// TIA Portal project "BOMBAS" (V15.1)

(* hardware
DEVICE "S7-1200 station_1"  S7-1200 Station
   slot 0: "Rack_0"  S7-1200 Rack  Rack  V1.0
   slot 1: "PLC_1"  CPU 1214C DC/DC/DC  6ES7 214-1AG40-0XB0  V4.2
DEVICE "HMI_1"  TP900 Comfort
   slot 0: "HMI_1"  TP900 Comfort  6AV2 124-0JC01-0AX0  15.1.0.0
   slot 1: "HMI_RT_1"  TP900 Comfort  6AV2 124-0JC01-0AX0  15.1.0.0
   slot 5: "HMI_1.IE_CP_1"  PROFINET Interface  15.0.1.0
      slot 1: "Interfaz PROFINET_1"  PROFINET Interface
         slot 1: "Port_1"  Port
         slot 2: "Port_2"  Port
   slot 7: "HMI_1.MPI/DP_CP_1"  MPI/DP Interface  15.0.1.0
*)

// ===== PLC "PLC_1"  CPU 1214C DC/DC/DC =====

VAR_GLOBAL   // PLC tag table "MODOS_ESTADOS"
   "HMI_PULSADOR_AUTOMATICO" AT %M2.1 : Bool;
   "HMI_PULSADOR_MANUAL" AT %M2.2 : Bool;
   "HMI_PULSADOR_STOP" AT %M2.3 : Bool;
   "ESTADO_MODO_MANUAL" AT %M2.4 : Bool;
   "ESTADO_MODO_AUTOMATICO" AT %M2.5 : Bool;
   "ESTADO_MODO_STOP" AT %M2.6 : Bool;
   "MODO_AUTOMATICO_START" AT %M2.7 : Bool;
   "HMI_PULSADOR_START" AT %M3.0 : Bool;
END_VAR

TYPE "BOMBA"
   STRUCT
      MOTOR : Bool;
      Tiempo_Total : UDInt;
      Tiempo_Acumulado : UDInt;
      Tiempo_Actual : UDInt;
      Tiempo_Trabajo : UDInt := 180;
   END_STRUCT;
END_TYPE

DATA_BLOCK "MAQUINA_ESTADO_BOMBAS_DB"   // DB1
{ S7_Optimized_Access := 'TRUE' }
VERSION : 0.1
// stored: InstanceOfName MAQUINA_ESTADO_BOMBAS
"MAQUINA_ESTADO_BOMBAS"
BEGIN
END_DATA_BLOCK

DATA_BLOCK "VARIABLES_GLOBALES"   // DB2
{ S7_Optimized_Access := 'TRUE' }
VERSION : 0.1
   VAR
      SALIDA_BOMBA_1 : "BOMBA";
      SALIDA_BOMBA_2 : "BOMBA";
      SALIDA_AUTOMATICO_BOMBA_1 : Bool;
      SALIDA_AUTOMATICO_BOMBA_2 : Bool;
      Tiempo_Cumplido_Bomba_1 : Bool;
      Tiempo_Cumplido_Bomba_2 : Bool;
      Tiempo_Formateado : Array[0..1] of Time_Of_Day;
      Numero_Str : String;
      HORA_STR : String;
      Tiempo_Bomba_1Str : String;
      Tiempo_Bomba_2Str : String;
      Variable_Ejemplo_VisualBasic : Int := 123;
      variable_string_visual : String := '123A';
      variable_string_visual2 : Array[0..2] of String;
      ejemplo_timeofdaytodint : DInt;
      tiempo : Time_Of_Day;
      Resultado_Conversion : Real;
   END_VAR
BEGIN
   SALIDA_BOMBA_1.Tiempo_Trabajo := 180;
   SALIDA_BOMBA_2.Tiempo_Trabajo := 180;
END_DATA_BLOCK

DATA_BLOCK "SALIDA_BOMBA_DB"   // DB3
{ S7_Optimized_Access := 'TRUE' }
VERSION : 0.1
// stored: InstanceOfName SALIDA_BOMBA
"SALIDA_BOMBA"
BEGIN
END_DATA_BLOCK

DATA_BLOCK "SALIDA_BOMBA_DB_1"   // DB5
{ S7_Optimized_Access := 'TRUE' }
VERSION : 0.1
// stored: InstanceOfName SALIDA_BOMBA
"SALIDA_BOMBA"
BEGIN
END_DATA_BLOCK

DATA_BLOCK "ALARMAS_DIAS"   // DB6
{ S7_Optimized_Access := 'TRUE' }
VERSION : 0.1
   VAR
      MOTORES : Array[1..3] of Struct
         DIA : Struct
            HORA_ACTIVACION : Array[1..7] of Time_Of_Day;
            HORA_DESACTIVACION : Array[1..7] of Time_Of_Day;
         END_STRUCT;
         ESTADO_MOTOR : Bool;
      END_STRUCT;
      HORA_ACTIVACION : Time_Of_Day;
      HORA_DESACTIVACION : Time_Of_Day;
   END_VAR
BEGIN
END_DATA_BLOCK

// folder: RELOJ

DATA_BLOCK "RELOJ_VARIABLES"   // DB4
{ S7_Optimized_Access := 'TRUE' }
VERSION : 0.1
   VAR
      HORA_ACTUAL : DTL;
      HORA_ANTERIOR : DTL;
      RET : Int;
      output_second : Bool;
   END_VAR
BEGIN
END_DATA_BLOCK

// folder: (top level)

FUNCTION_BLOCK "MAQUINA_ESTADO_BOMBAS"   // FB1, SCL
{ S7_Optimized_Access := 'TRUE' }
VERSION : 0.1
   VAR_INPUT
      ESTADO_AUTOMATICO : Bool;
      BOTON_START : Bool;
      BOTON_PARO_AUTOMATICO : Bool;
      Tiempo_Cumplido_Bomba_1 : Bool;
      Tiempo_Cumplido_Bomba_2 : Bool;
      BOTON_PARO_GENERAL : Bool;
      Tiempo_Bomba_1 : UDInt;
      Tiempo_Bomba_2 : UDInt;
   END_VAR
   VAR_OUTPUT
      MOTOR1 : Bool;
      MOTOR2 : Bool;
   END_VAR
   VAR
      ESTADO : USInt := 0;
   END_VAR
   VAR CONSTANT
      ESTADO_0 : USInt := 0;
      ESTADO_1 : USInt := 1;
      ESTADO_2 : USInt := 2;
      ESTADO_3 : USInt := 3;
      ESTADO_4 : USInt := 4;
      ESTADO_5 : USInt := 5;
      ESTADO_6 : USInt := 6;
      ESTADO_7 : USInt := 7;
      ESTADO_8 : USInt := 8;
      ESTADO_9 : USInt := 9;
   END_VAR
BEGIN
   // ESTADOS ENTRADAS
   CASE #ESTADO OF
       #ESTADO_0:  // Statement section case 1
           IF #ESTADO_AUTOMATICO THEN
               #ESTADO := #ESTADO_1;
           END_IF;
       #ESTADO_1:  // Statement section case 2 to 4
           IF #BOTON_START THEN
               #ESTADO := #ESTADO_2;
           END_IF;
           IF #BOTON_PARO_GENERAL THEN
               #ESTADO := #ESTADO_0;
           END_IF;
       #ESTADO_2:  // Statement section case 2 to 4
           IF #Tiempo_Bomba_1<=#Tiempo_Bomba_2 THEN
               #ESTADO := #ESTADO_3;
           ELSE
               #ESTADO := #ESTADO_5;
           END_IF;
           IF #BOTON_PARO_GENERAL THEN
               #ESTADO := #ESTADO_0;
           END_IF;
       #ESTADO_3:
           IF #Tiempo_Cumplido_Bomba_1 THEN
               #ESTADO := #ESTADO_4;
           END_IF;
           IF #BOTON_PARO_GENERAL THEN
               #ESTADO := #ESTADO_0;
           END_IF;
       #ESTADO_4:
           IF #Tiempo_Cumplido_Bomba_2 THEN
               #ESTADO := #ESTADO_3;
           END_IF;
           IF #BOTON_PARO_GENERAL THEN
               #ESTADO := #ESTADO_0;
           END_IF;
       #ESTADO_5:
           IF #Tiempo_Cumplido_Bomba_2 THEN
               #ESTADO := #ESTADO_6;
           END_IF;
           IF #BOTON_PARO_GENERAL THEN
               #ESTADO := #ESTADO_0;
           END_IF;
       #ESTADO_6:
           IF #Tiempo_Cumplido_Bomba_1 THEN
               #ESTADO := #ESTADO_5;
           END_IF;
           IF #BOTON_PARO_GENERAL THEN
               #ESTADO := #ESTADO_0;
           END_IF;
       ELSE  // Statement section ELSE
           ;
   END_CASE;
   //ESTADOS_SALIDAS
   CASE #ESTADO OF
       #ESTADO_0:  // Statement section case 1
           #MOTOR1 := FALSE;
           #MOTOR2 := FALSE;
       #ESTADO_1:  // Statement section case 2 to 4
           ;
       #ESTADO_2:
           ;
       #ESTADO_3:
           #MOTOR2 := FALSE;
           #MOTOR1 := TRUE;
       #ESTADO_4:
           #MOTOR2 := TRUE;
           #MOTOR1 := FALSE;
       #ESTADO_5:
           #MOTOR2 := TRUE;
           #MOTOR1 := FALSE;
       #ESTADO_6:
           #MOTOR2 := FALSE;
           #MOTOR1 := TRUE;
       #ESTADO_7:
           ;
   END_CASE;
END_FUNCTION_BLOCK

FUNCTION_BLOCK "SALIDA_BOMBA"   // FB2, SCL
{ S7_Optimized_Access := 'TRUE' }
VERSION : 0.1
   VAR_INPUT
      Entrada_Segundo : Bool;
   END_VAR
   VAR_OUTPUT
      Tiempo_Cumplido_Bomba : Bool;
      Tiempo_Total_TimeofDa : Time_Of_Day;
   END_VAR
   VAR_IN_OUT
      ENTRADA_BOMBA : "BOMBA";
   END_VAR
BEGIN
   #ENTRADA_BOMBA.Tiempo_Trabajo := 180;
   IF NOT #ENTRADA_BOMBA.MOTOR THEN
       #ENTRADA_BOMBA.Tiempo_Acumulado := 0;
   END_IF;
   IF #Entrada_Segundo AND #ENTRADA_BOMBA.MOTOR THEN
       #ENTRADA_BOMBA.Tiempo_Actual :=1;
       #ENTRADA_BOMBA.Tiempo_Acumulado := #ENTRADA_BOMBA.Tiempo_Acumulado + 1;
       #ENTRADA_BOMBA.Tiempo_Total := #ENTRADA_BOMBA.Tiempo_Actual + #ENTRADA_BOMBA.Tiempo_Total;
   END_IF;
   IF #ENTRADA_BOMBA.Tiempo_Acumulado >= #ENTRADA_BOMBA.Tiempo_Trabajo THEN
       #ENTRADA_BOMBA.Tiempo_Actual := 0;
       #Tiempo_Cumplido_Bomba := true;
       #ENTRADA_BOMBA.Tiempo_Acumulado := 0;
   ELSE
       #Tiempo_Cumplido_Bomba := false;
   END_IF;
   #Tiempo_Total_TimeofDa:= UDINT_TO_TOD(#ENTRADA_BOMBA.Tiempo_Total+10000);
END_FUNCTION_BLOCK

FUNCTION "US_TIMEOFDAY" : Void   // FC2, SCL
{ S7_Optimized_Access := 'TRUE' }
VERSION : 0.1
   VAR_INPUT
      SEGUNDOS : UDInt;
   END_VAR
   VAR_OUTPUT
      string_output : String;
   END_VAR
   VAR_TEMP
      str_horas : String;
      str_minutos : String;
      str_segundos : String;
      str_output : String;
      Horas : UDInt;
      Minutos : UDInt;
      Segundos_1 : UDInt;
   END_VAR
   VAR CONSTANT
      const_horas : UDInt := 3600;
      const_minutos : UDInt := 60;
   END_VAR
BEGIN
   #Horas := #SEGUNDOS / 3600;
   #Minutos := (#SEGUNDOS MOD 3600) / 60;
   #Segundos_1 := ((#SEGUNDOS MOD 3600)MOD 60);
   "US_TOSTRING"(Numero:=#Horas,
                 output=>#str_horas);
   "US_TOSTRING"(Numero := #Minutos,
                 output => #str_minutos);
   "US_TOSTRING"(Numero := #Segundos_1,
                 output => #str_segundos);


   #str_output:= CONCAT(IN1 := #str_output, IN2 := #str_horas,IN3:=':'
                        ,IN4:=#str_minutos,IN5:=':',IN6:=#str_segundos);
   #string_output := #str_output;
END_FUNCTION

FUNCTION "US_TOSTRING" : Void   // FC3, SCL
{ S7_Optimized_Access := 'TRUE' }
VERSION : 0.1
   VAR_INPUT
      Numero : UDInt;
   END_VAR
   VAR_OUTPUT
      output : String;
   END_VAR
   VAR_TEMP
      contador : USInt;
      Arreglo : Array[0..3] of Char;
      centenas : UDInt;
      decenas : UDInt;
      unidades : UDInt;
   END_VAR
BEGIN
   #contador := 0;
   #centenas := #Numero / 100;
   #decenas := (#Numero MOD 100)/10;
   #unidades := (#Numero MOD 100) MOD 10;
   IF #centenas <> 0 THEN
       CASE #centenas OF
           0:
               #Arreglo[#contador] := '0';
           1:  // Statement section case 1
               #Arreglo[#contador] := '1';
           2:  // Statement section case 2 to 4
               #Arreglo[#contador] := '2';
           3:
               #Arreglo[#contador] := '3';
           4:
               #Arreglo[#contador] := '4';
           5:
               #Arreglo[#contador] := '5';
           6:
               #Arreglo[#contador] := '6';
           7:
               #Arreglo[#contador] := '7';
           8:
               #Arreglo[#contador] := '8';
           9:
               #Arreglo[#contador] := '9';
       END_CASE;
       #contador := #contador + 1;
   END_IF;
       CASE #decenas OF
           0:
               #Arreglo[#contador] := '0';
           1:  // Statement section case 1
               #Arreglo[#contador] := '1';
           2:  // Statement section case 2 to 4
               #Arreglo[#contador] := '2';
           3:
               #Arreglo[#contador] := '3';
           4:
               #Arreglo[#contador] := '4';
           5:
               #Arreglo[#contador] := '5';
           6:
               #Arreglo[#contador] := '6';
           7:
               #Arreglo[#contador] := '7';
           8:
               #Arreglo[#contador] := '8';
           9:
               #Arreglo[#contador] := '9';
       END_CASE;
       #contador := #contador + 1;
       CASE #unidades OF
           0:
               #Arreglo[#contador] := '0';
           1:  // Statement section case 1
               #Arreglo[#contador] := '1';
           2:  // Statement section case 2 to 4
               #Arreglo[#contador] := '2';
           3:
               #Arreglo[#contador] := '3';
           4:
               #Arreglo[#contador] := '4';
           5:
               #Arreglo[#contador] := '5';
           6:
               #Arreglo[#contador] := '6';
           7:
               #Arreglo[#contador] := '7';
           8:
               #Arreglo[#contador] := '8';
           9:
               #Arreglo[#contador] := '9';
       END_CASE;
       #contador := #contador + 1;
   Chars_TO_Strg(Chars:=#Arreglo,
                 pChars:=0,
                 Cnt:=#contador,
                 Strg=>#output);
END_FUNCTION

FUNCTION "CONVERTIR_DWORD_FLOAT" : Void   // FC4, SCL
{ S7_Optimized_Access := 'TRUE' }
VERSION : 0.1
   VAR_INPUT
      PARTE_ALTA : DWord;
      PARTE_BAJ : DWord;
   END_VAR
   VAR_OUTPUT
      Salida : Real;
   END_VAR
   VAR_TEMP
      TRAMA : DWord;
   END_VAR
BEGIN
   #TRAMA:=SHL(IN:=#PARTE_ALTA, N:=16) OR #PARTE_BAJ;
   #Salida:=DWORD_TO_REAL(#TRAMA);
END_FUNCTION

FUNCTION "Bloque_1" : Void   // FC5, SCL
{ S7_Optimized_Access := 'TRUE' }
VERSION : 0.1
   VAR_TEMP
      HORA_DIA : Time_Of_Day;
      FECHA_HOY : DTL;
      res : Int;
      i : Int;
   END_VAR
BEGIN
   #res := RD_LOC_T(#FECHA_HOY);
   #HORA_DIA := DTL_TO_TOD(#FECHA_HOY);
   FOR #i := 1 TO 3  BY 1 DO
       "ALARMAS_DIAS".HORA_ACTIVACION := "ALARMAS_DIAS".MOTORES[#i].DIA.HORA_ACTIVACION[#FECHA_HOY.WEEKDAY];
       "ALARMAS_DIAS".HORA_DESACTIVACION := "ALARMAS_DIAS".MOTORES[#i].DIA.HORA_DESACTIVACION[#FECHA_HOY.WEEKDAY];
       "ALARMAS_DIAS".MOTORES[#i].DIA.HORA_ACTIVACION[#FECHA_HOY.WEEKDAY] := "ALARMAS_DIAS".HORA_ACTIVACION;
       "ALARMAS_DIAS".MOTORES[#i].DIA.HORA_DESACTIVACION[#FECHA_HOY.WEEKDAY] := "ALARMAS_DIAS".HORA_DESACTIVACION;
       "ALARMAS_DIAS".MOTORES[#i].ESTADO_MOTOR := #HORA_DIA >= "ALARMAS_DIAS".HORA_ACTIVACION AND #HORA_DIA < "ALARMAS_DIAS".HORA_DESACTIVACION;
   END_FOR;
END_FUNCTION

ORGANIZATION_BLOCK "Main"   // OB1, LAD, ProgramCycle
TITLE = "Main Program Sweep (Cycle)"
{ S7_Optimized_Access := 'TRUE' }
VERSION : 0.1
   VAR_INPUT
      Initial_Call : Bool;   // Initial call of this OB
      Remanence : Bool;   // =True, if remanent data are available
   END_VAR
BEGIN

REGION Network 1: LEO_UN_SEGUNDO
   // LEO_UN_SEGUNDO
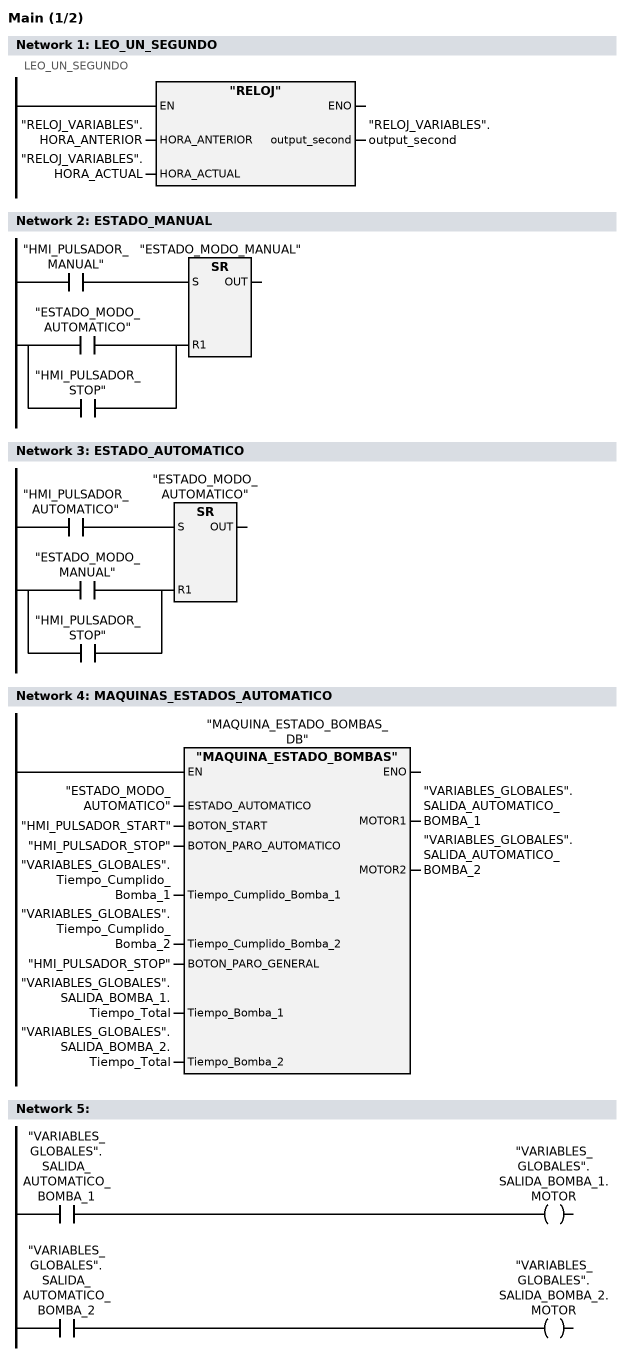
   RUNG wire#powerrail
      "RELOJ"(HORA_ANTERIOR := "RELOJ_VARIABLES".HORA_ANTERIOR, HORA_ACTUAL := "RELOJ_VARIABLES".HORA_ACTUAL, output_second => "RELOJ_VARIABLES".output_second)
   END_RUNG
   // the same network as SCL:
   "RELOJ"(HORA_ANTERIOR := "RELOJ_VARIABLES".HORA_ANTERIOR,
           HORA_ACTUAL := "RELOJ_VARIABLES".HORA_ACTUAL,
           output_second => "RELOJ_VARIABLES".output_second);
END_REGION

REGION Network 2: ESTADO_MANUAL
   RUNG wire#powerrail
      Contact( "HMI_PULSADOR_MANUAL" )
      S_SR(operand := "ESTADO_MODO_MANUAL", r1 := wire#w1)
   END_RUNG
   RUNG wire#powerrail
      Contact( "ESTADO_MODO_AUTOMATICO" )
   END_RUNG wire#w1
   RUNG wire#powerrail
      Contact( "HMI_PULSADOR_STOP" )
   END_RUNG wire#w1
   // the same network as SCL:
   IF "HMI_PULSADOR_MANUAL" THEN
       "ESTADO_MODO_MANUAL" := TRUE;   // SR flip-flop
   END_IF;
   IF "ESTADO_MODO_AUTOMATICO" OR "HMI_PULSADOR_STOP" THEN "ESTADO_MODO_MANUAL" := FALSE; END_IF;
END_REGION

REGION Network 3: ESTADO_AUTOMATICO
   RUNG wire#powerrail
      Contact( "HMI_PULSADOR_AUTOMATICO" )
      S_SR(operand := "ESTADO_MODO_AUTOMATICO", r1 := wire#w1)
   END_RUNG
   RUNG wire#powerrail
      Contact( "ESTADO_MODO_MANUAL" )
   END_RUNG wire#w1
   RUNG wire#powerrail
      Contact( "HMI_PULSADOR_STOP" )
   END_RUNG wire#w1
   // the same network as SCL:
   IF "HMI_PULSADOR_AUTOMATICO" THEN
       "ESTADO_MODO_AUTOMATICO" := TRUE;   // SR flip-flop
   END_IF;
   IF "ESTADO_MODO_MANUAL" OR "HMI_PULSADOR_STOP" THEN "ESTADO_MODO_AUTOMATICO" := FALSE; END_IF;
END_REGION

REGION Network 4: MAQUINAS_ESTADOS_AUTOMATICO
   RUNG wire#powerrail
      "MAQUINA_ESTADO_BOMBAS_DB"(ESTADO_AUTOMATICO := "ESTADO_MODO_AUTOMATICO", BOTON_START := "HMI_PULSADOR_START", BOTON_PARO_AUTOMATICO := "HMI_PULSADOR_STOP", Tiempo_Cumplido_Bomba_1 := "VARIABLES_GLOBALES".Tiempo_Cumplido_Bomba_1, Tiempo_Cumplido_Bomba_2 := "VARIABLES_GLOBALES".Tiempo_Cumplido_Bomba_2, BOTON_PARO_GENERAL := "HMI_PULSADOR_STOP", Tiempo_Bomba_1 := "VARIABLES_GLOBALES".SALIDA_BOMBA_1.Tiempo_Total, Tiempo_Bomba_2 := "VARIABLES_GLOBALES".SALIDA_BOMBA_2.Tiempo_Total, MOTOR1 => "VARIABLES_GLOBALES".SALIDA_AUTOMATICO_BOMBA_1, MOTOR2 => "VARIABLES_GLOBALES".SALIDA_AUTOMATICO_BOMBA_2)
   END_RUNG
   // the same network as SCL:
   "MAQUINA_ESTADO_BOMBAS_DB"(ESTADO_AUTOMATICO := "ESTADO_MODO_AUTOMATICO",   // "MAQUINA_ESTADO_BOMBAS"
                           BOTON_START := "HMI_PULSADOR_START",
                           BOTON_PARO_AUTOMATICO := "HMI_PULSADOR_STOP",
                           Tiempo_Cumplido_Bomba_1 := "VARIABLES_GLOBALES".Tiempo_Cumplido_Bomba_1,
                           Tiempo_Cumplido_Bomba_2 := "VARIABLES_GLOBALES".Tiempo_Cumplido_Bomba_2,
                           BOTON_PARO_GENERAL := "HMI_PULSADOR_STOP",
                           Tiempo_Bomba_1 := "VARIABLES_GLOBALES".SALIDA_BOMBA_1.Tiempo_Total,
                           Tiempo_Bomba_2 := "VARIABLES_GLOBALES".SALIDA_BOMBA_2.Tiempo_Total,
                           MOTOR1 => "VARIABLES_GLOBALES".SALIDA_AUTOMATICO_BOMBA_1,
                           MOTOR2 => "VARIABLES_GLOBALES".SALIDA_AUTOMATICO_BOMBA_2);
END_REGION

REGION Network 5
   RUNG wire#powerrail
      Contact( "VARIABLES_GLOBALES".SALIDA_AUTOMATICO_BOMBA_1 )
      Coil( "VARIABLES_GLOBALES".SALIDA_BOMBA_1.MOTOR )
   END_RUNG
   RUNG wire#powerrail
      Contact( "VARIABLES_GLOBALES".SALIDA_AUTOMATICO_BOMBA_2 )
      Coil( "VARIABLES_GLOBALES".SALIDA_BOMBA_2.MOTOR )
   END_RUNG
   // the same network as SCL:
   "VARIABLES_GLOBALES".SALIDA_BOMBA_1.MOTOR := "VARIABLES_GLOBALES".SALIDA_AUTOMATICO_BOMBA_1;
   "VARIABLES_GLOBALES".SALIDA_BOMBA_2.MOTOR := "VARIABLES_GLOBALES".SALIDA_AUTOMATICO_BOMBA_2;
END_REGION

REGION Network 6: SALIDA_MOTOR1_
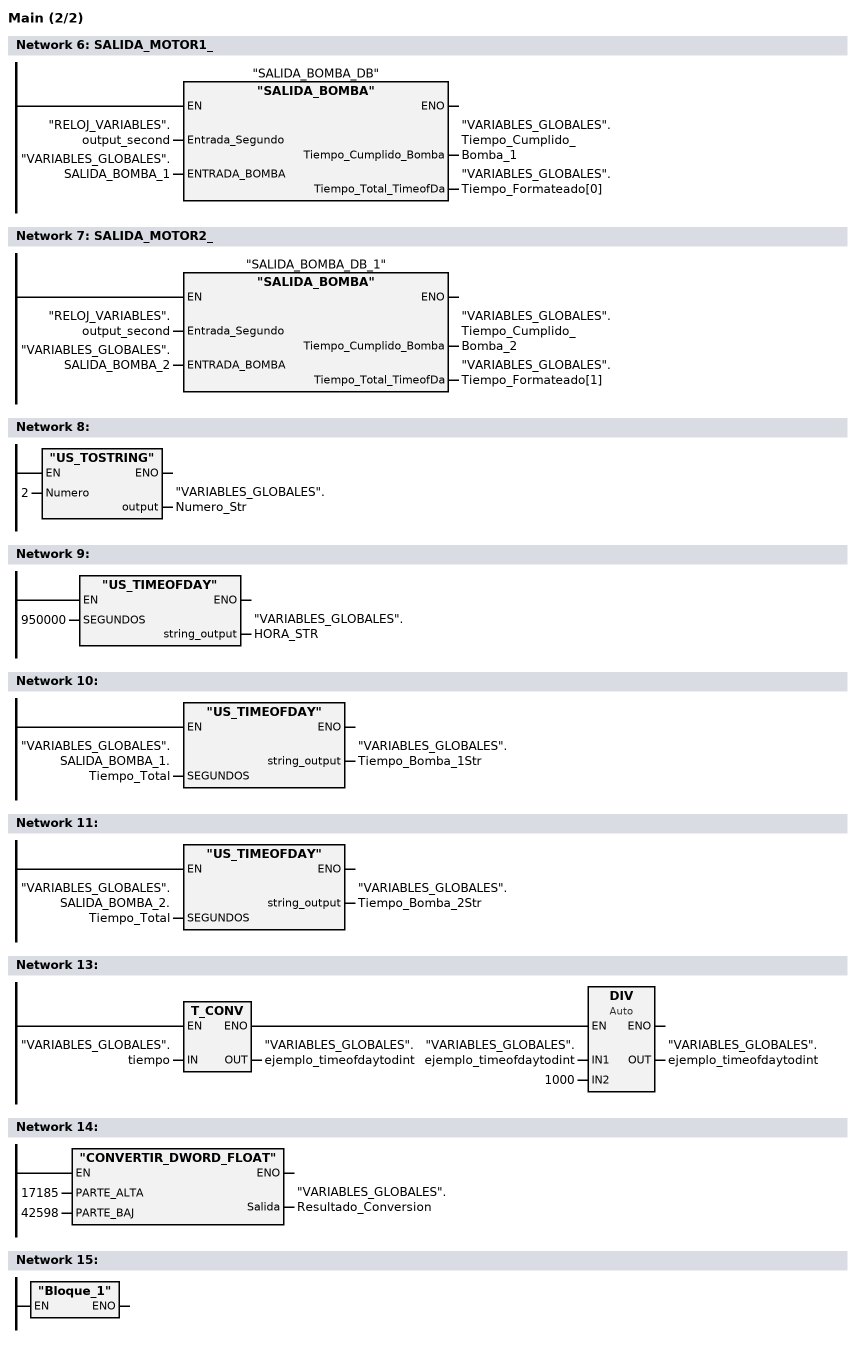
   RUNG wire#powerrail
      "SALIDA_BOMBA_DB"(Entrada_Segundo := "RELOJ_VARIABLES".output_second, ENTRADA_BOMBA := "VARIABLES_GLOBALES".SALIDA_BOMBA_1, Tiempo_Cumplido_Bomba => "VARIABLES_GLOBALES".Tiempo_Cumplido_Bomba_1, Tiempo_Total_TimeofDa => "VARIABLES_GLOBALES".Tiempo_Formateado[0])
   END_RUNG
   // the same network as SCL:
   "SALIDA_BOMBA_DB"(Entrada_Segundo := "RELOJ_VARIABLES".output_second,   // "SALIDA_BOMBA"
                     ENTRADA_BOMBA := "VARIABLES_GLOBALES".SALIDA_BOMBA_1,
                     Tiempo_Cumplido_Bomba => "VARIABLES_GLOBALES".Tiempo_Cumplido_Bomba_1,
                     Tiempo_Total_TimeofDa => "VARIABLES_GLOBALES".Tiempo_Formateado[0]);
END_REGION

REGION Network 7: SALIDA_MOTOR2_
   RUNG wire#powerrail
      "SALIDA_BOMBA_DB_1"(Entrada_Segundo := "RELOJ_VARIABLES".output_second, ENTRADA_BOMBA := "VARIABLES_GLOBALES".SALIDA_BOMBA_2, Tiempo_Cumplido_Bomba => "VARIABLES_GLOBALES".Tiempo_Cumplido_Bomba_2, Tiempo_Total_TimeofDa => "VARIABLES_GLOBALES".Tiempo_Formateado[1])
   END_RUNG
   // the same network as SCL:
   "SALIDA_BOMBA_DB_1"(Entrada_Segundo := "RELOJ_VARIABLES".output_second,   // "SALIDA_BOMBA"
                       ENTRADA_BOMBA := "VARIABLES_GLOBALES".SALIDA_BOMBA_2,
                       Tiempo_Cumplido_Bomba => "VARIABLES_GLOBALES".Tiempo_Cumplido_Bomba_2,
                       Tiempo_Total_TimeofDa => "VARIABLES_GLOBALES".Tiempo_Formateado[1]);
END_REGION

REGION Network 8
   RUNG wire#powerrail
      "US_TOSTRING"(Numero := 2, output => "VARIABLES_GLOBALES".Numero_Str)
   END_RUNG
   // the same network as SCL:
   "US_TOSTRING"(Numero := 2, output => "VARIABLES_GLOBALES".Numero_Str);
END_REGION

REGION Network 9
   RUNG wire#powerrail
      "US_TIMEOFDAY"(SEGUNDOS := 950000, string_output => "VARIABLES_GLOBALES".HORA_STR)
   END_RUNG
   // the same network as SCL:
   "US_TIMEOFDAY"(SEGUNDOS := 950000, string_output => "VARIABLES_GLOBALES".HORA_STR);
END_REGION

REGION Network 10
   RUNG wire#powerrail
      "US_TIMEOFDAY"(SEGUNDOS := "VARIABLES_GLOBALES".SALIDA_BOMBA_1.Tiempo_Total, string_output => "VARIABLES_GLOBALES".Tiempo_Bomba_1Str)
   END_RUNG
   // the same network as SCL:
   "US_TIMEOFDAY"(SEGUNDOS := "VARIABLES_GLOBALES".SALIDA_BOMBA_1.Tiempo_Total,
                  string_output => "VARIABLES_GLOBALES".Tiempo_Bomba_1Str);
END_REGION

REGION Network 11
   RUNG wire#powerrail
      "US_TIMEOFDAY"(SEGUNDOS := "VARIABLES_GLOBALES".SALIDA_BOMBA_2.Tiempo_Total, string_output => "VARIABLES_GLOBALES".Tiempo_Bomba_2Str)
   END_RUNG
   // the same network as SCL:
   "US_TIMEOFDAY"(SEGUNDOS := "VARIABLES_GLOBALES".SALIDA_BOMBA_2.Tiempo_Total,
                  string_output => "VARIABLES_GLOBALES".Tiempo_Bomba_2Str);
END_REGION

REGION Network 13
   // ENO of a box is taken as its EN; it also drops when the box reports an error
   "VARIABLES_GLOBALES".ejemplo_timeofdaytodint := T_CONV(IN := "VARIABLES_GLOBALES".tiempo);
   "VARIABLES_GLOBALES".ejemplo_timeofdaytodint := "VARIABLES_GLOBALES".ejemplo_timeofdaytodint / 1000;
END_REGION

REGION Network 14
   RUNG wire#powerrail
      "CONVERTIR_DWORD_FLOAT"(PARTE_ALTA := 17185, PARTE_BAJ := 42598, Salida => "VARIABLES_GLOBALES".Resultado_Conversion)
   END_RUNG
   // the same network as SCL:
   "CONVERTIR_DWORD_FLOAT"(PARTE_ALTA := 17185,
                           PARTE_BAJ := 42598,
                           Salida => "VARIABLES_GLOBALES".Resultado_Conversion);
END_REGION

REGION Network 15
   RUNG wire#powerrail
      "Bloque_1"()
   END_RUNG
   // the same network as SCL:
   "Bloque_1"();
END_REGION
END_ORGANIZATION_BLOCK

// folder: RELOJ

FUNCTION "RELOJ" : Void   // FC1, SCL
{ S7_Optimized_Access := 'TRUE' }
VERSION : 0.1
   VAR_OUTPUT
      output_second : Bool;
   END_VAR
   VAR_IN_OUT
      HORA_ANTERIOR : DTL;
      HORA_ACTUAL : DTL;
   END_VAR
   VAR_TEMP
      RET : Int;
   END_VAR
BEGIN
   #RET:=RD_SYS_T(#HORA_ACTUAL);
   #output_second := #HORA_ACTUAL.SECOND <> #HORA_ANTERIOR.SECOND ;
   #HORA_ANTERIOR := #HORA_ACTUAL;
END_FUNCTION

(* ===== HMI "HMI_RT_1" =====
system functions are stored by id; their names below are inferred from use
connection "HMI_Conexión_1": ETHERNET, S7_1200_OMS

HMI tags "Tabla de variables estándar"
   "Número_imagen_variable" : UInt, internal
   "ESTADO_MODO_AUTOMATICO" : Bool = PLC ESTADO_MODO_AUTOMATICO AT %M2.5, 100 ms
   "HMI_PULSADOR_AUTOMATICO" : Bool = PLC HMI_PULSADOR_AUTOMATICO AT %M2.1, 100 ms
   "HMI_PULSADOR_START" : Bool = PLC HMI_PULSADOR_START AT %M3.0, 100 ms
   "VARIABLES_GLOBALES_SALIDA_AUTOMATICO_BOMBA_1" : Bool = PLC VARIABLES_GLOBALES.SALIDA_AUTOMATICO_BOMBA_1, 100 ms
   "VARIABLES_GLOBALES_SALIDA_AUTOMATICO_BOMBA_2" : Bool = PLC VARIABLES_GLOBALES.SALIDA_AUTOMATICO_BOMBA_2, 100 ms
   "VARIABLES_GLOBALES_HORA_STR" : String[254] = PLC VARIABLES_GLOBALES.HORA_STR, 100 ms
   "HMI_PULSADOR_STOP" : Bool = PLC HMI_PULSADOR_STOP AT %M2.3, 100 ms
   "VARIABLES_GLOBALES_Tiempo_Bomba_1Str" : String[254] = PLC VARIABLES_GLOBALES.Tiempo_Bomba_1Str, 100 ms
   "VARIABLES_GLOBALES_Tiempo_Bomba_2Str" : String[254] = PLC VARIABLES_GLOBALES.Tiempo_Bomba_2Str, 100 ms
   "VARIABLES_GLOBALES_Variable_Ejemplo_VisualBasic_2" : Int = PLC VARIABLES_GLOBALES.Variable_Ejemplo_VisualBasic AT %DB1.DBW0, 100 ms
   "VARIABLES_GLOBALES_variable_string_visual" : String[254] = PLC VARIABLES_GLOBALES.variable_string_visual, 100 ms
   "VARIABLES_GLOBALES_variable_string_visual2{0}" : String[254] = PLC VARIABLES_GLOBALES.variable_string_visual2[0], 100 ms
   "VARIABLES_GLOBALES_tiempo" : Time_Of_Day = PLC VARIABLES_GLOBALES.tiempo, 100 ms
   "ALARMAS_DIAS_MOTORES{1}_DIA_HORA_ACTIVACION{1}" : Time_Of_Day = PLC ALARMAS_DIAS.MOTORES[1].DIA.HORA_ACTIVACION[1], 1 s
   "ALARMAS_DIAS_MOTORES{1}_DIA_HORA_DESACTIVACION{1}" : Time_Of_Day = PLC ALARMAS_DIAS.MOTORES[1].DIA.HORA_DESACTIVACION[1], 1 s
   "ALARMAS_DIAS_MOTORES{1}_DIA_HORA_ACTIVACION{2}" : Time_Of_Day = PLC ALARMAS_DIAS.MOTORES[1].DIA.HORA_ACTIVACION[2], 1 s
   "ALARMAS_DIAS_MOTORES{1}_DIA_HORA_DESACTIVACION{2}" : Time_Of_Day = PLC ALARMAS_DIAS.MOTORES[1].DIA.HORA_DESACTIVACION[2], 1 s
   "ALARMAS_DIAS_MOTORES{1}_DIA_HORA_DESACTIVACION{3}" : Time_Of_Day = PLC ALARMAS_DIAS.MOTORES[1].DIA.HORA_DESACTIVACION[3], 1 s
   "ALARMAS_DIAS_MOTORES{1}_DIA_HORA_ACTIVACION{3}" : Time_Of_Day = PLC ALARMAS_DIAS.MOTORES[1].DIA.HORA_ACTIVACION[3], 1 s
   "ALARMAS_DIAS_MOTORES{1}_DIA_HORA_ACTIVACION{4}" : Time_Of_Day = PLC ALARMAS_DIAS.MOTORES[1].DIA.HORA_ACTIVACION[4], 1 s
   "ALARMAS_DIAS_MOTORES{1}_DIA_HORA_ACTIVACION{5}" : Time_Of_Day = PLC ALARMAS_DIAS.MOTORES[1].DIA.HORA_ACTIVACION[5], 1 s
   "ALARMAS_DIAS_MOTORES{1}_DIA_HORA_ACTIVACION{6}" : Time_Of_Day = PLC ALARMAS_DIAS.MOTORES[1].DIA.HORA_ACTIVACION[6], 1 s
   "ALARMAS_DIAS_MOTORES{1}_DIA_HORA_ACTIVACION{7}" : Time_Of_Day = PLC ALARMAS_DIAS.MOTORES[1].DIA.HORA_ACTIVACION[7], 1 s
   "ALARMAS_DIAS_MOTORES{1}_DIA_HORA_DESACTIVACION{4}" : Time_Of_Day = PLC ALARMAS_DIAS.MOTORES[1].DIA.HORA_DESACTIVACION[4], 1 s
   "ALARMAS_DIAS_MOTORES{1}_DIA_HORA_DESACTIVACION{5}" : Time_Of_Day = PLC ALARMAS_DIAS.MOTORES[1].DIA.HORA_DESACTIVACION[5], 1 s
   "ALARMAS_DIAS_MOTORES{1}_DIA_HORA_DESACTIVACION{6}" : Time_Of_Day = PLC ALARMAS_DIAS.MOTORES[1].DIA.HORA_DESACTIVACION[6], 1 s
   "ALARMAS_DIAS_MOTORES{1}_DIA_HORA_DESACTIVACION{7}" : Time_Of_Day = PLC ALARMAS_DIAS.MOTORES[1].DIA.HORA_DESACTIVACION[7], 1 s
   "ALARMAS_DIAS_MOTORES{1}_ESTADO_MOTOR" : Bool = PLC ALARMAS_DIAS.MOTORES[1].ESTADO_MOTOR, 1 s
   "ALARMAS_DIAS_MOTORES{2}_ESTADO_MOTOR" : Bool = PLC ALARMAS_DIAS.MOTORES[2].ESTADO_MOTOR, 1 s
   "ALARMAS_DIAS_MOTORES{2}_DIA_HORA_ACTIVACION{1}" : Time_Of_Day = PLC ALARMAS_DIAS.MOTORES[2].DIA.HORA_ACTIVACION[1], 1 s
   "ALARMAS_DIAS_MOTORES{2}_DIA_HORA_ACTIVACION{2}" : Time_Of_Day = PLC ALARMAS_DIAS.MOTORES[2].DIA.HORA_ACTIVACION[2], 1 s
   "ALARMAS_DIAS_MOTORES{2}_DIA_HORA_ACTIVACION{3}" : Time_Of_Day = PLC ALARMAS_DIAS.MOTORES[2].DIA.HORA_ACTIVACION[3], 1 s
   "ALARMAS_DIAS_MOTORES{2}_DIA_HORA_ACTIVACION{4}" : Time_Of_Day = PLC ALARMAS_DIAS.MOTORES[2].DIA.HORA_ACTIVACION[4], 1 s
   "ALARMAS_DIAS_MOTORES{2}_DIA_HORA_ACTIVACION{5}" : Time_Of_Day = PLC ALARMAS_DIAS.MOTORES[2].DIA.HORA_ACTIVACION[5], 1 s
   "ALARMAS_DIAS_MOTORES{2}_DIA_HORA_ACTIVACION{6}" : Time_Of_Day = PLC ALARMAS_DIAS.MOTORES[2].DIA.HORA_ACTIVACION[6], 1 s
   "ALARMAS_DIAS_MOTORES{2}_DIA_HORA_ACTIVACION{7}" : Time_Of_Day = PLC ALARMAS_DIAS.MOTORES[2].DIA.HORA_ACTIVACION[7], 1 s
   "ALARMAS_DIAS_MOTORES{2}_DIA_HORA_DESACTIVACION{1}" : Time_Of_Day = PLC ALARMAS_DIAS.MOTORES[2].DIA.HORA_DESACTIVACION[1], 1 s
   "ALARMAS_DIAS_MOTORES{2}_DIA_HORA_DESACTIVACION{2}" : Time_Of_Day = PLC ALARMAS_DIAS.MOTORES[2].DIA.HORA_DESACTIVACION[2], 1 s
   "ALARMAS_DIAS_MOTORES{2}_DIA_HORA_DESACTIVACION{3}" : Time_Of_Day = PLC ALARMAS_DIAS.MOTORES[2].DIA.HORA_DESACTIVACION[3], 1 s
   "ALARMAS_DIAS_MOTORES{2}_DIA_HORA_DESACTIVACION{4}" : Time_Of_Day = PLC ALARMAS_DIAS.MOTORES[2].DIA.HORA_DESACTIVACION[4], 1 s
   "ALARMAS_DIAS_MOTORES{2}_DIA_HORA_DESACTIVACION{5}" : Time_Of_Day = PLC ALARMAS_DIAS.MOTORES[2].DIA.HORA_DESACTIVACION[5], 1 s
   "ALARMAS_DIAS_MOTORES{2}_DIA_HORA_DESACTIVACION{6}" : Time_Of_Day = PLC ALARMAS_DIAS.MOTORES[2].DIA.HORA_DESACTIVACION[6], 1 s
   "ALARMAS_DIAS_MOTORES{2}_DIA_HORA_DESACTIVACION{7}" : Time_Of_Day = PLC ALARMAS_DIAS.MOTORES[2].DIA.HORA_DESACTIVACION[7], 1 s

text list "Nombre_imagen_lista_texto": 1 'Imagen raíz'

screen "Imagen raíz" 800x420, template "Plantilla_1"
   on GenerateScreen: SetTag("Número_imagen_variable", 1)
   Button "Botón_1" at 52,44 size 96x32; TextOff 'Text'
      on Press: SetBit("HMI_PULSADOR_AUTOMATICO"); "FuncionVB_1"()
      on Release: ResetBit("HMI_PULSADOR_AUTOMATICO")
   Button "Botón_2" at 55,96 size 96x32; TextOff 'Text'
      on Press: SetBit("HMI_PULSADOR_START")
      on Release: ResetBit("HMI_PULSADOR_START")
   SymbolLibrary "Librería de símbolos_1" at 309,122 size 36x31
      Appearance <- "VARIABLES_GLOBALES_SALIDA_AUTOMATICO_BOMBA_1"
   SymbolLibrary "Librería de símbolos_2" at 285,274 size 46x46
      Appearance <- "VARIABLES_GLOBALES_SALIDA_AUTOMATICO_BOMBA_2"
   IOField "Campo ES_1" at 395,69 size 82x32; FormatPattern ????????????????????????????????????????????????????????????????????????????????
      ProcessValue <- "VARIABLES_GLOBALES_HORA_STR"
   Button "Botón_3" at 52,157 size 96x32; TextOff 'Text'
      on Release: ResetBit("HMI_PULSADOR_STOP")
      on Press: SetBit("HMI_PULSADOR_STOP")
   IOField "Campo ES_2" at 342,258 size 89x29; FormatPattern ????????????????????????????????????????????????????????????????????????????????
      ProcessValue <- "VARIABLES_GLOBALES_Tiempo_Bomba_1Str"
   IOField "Campo ES_3" at 607,258 size 82x32; FormatPattern ????????????????????????????????????????????????????????????????????????????????
      ProcessValue <- "VARIABLES_GLOBALES_Tiempo_Bomba_2Str"
   IOField "Campo ES_4" at 464,121 size 82x32; FormatPattern s99999
      ProcessValue <- "VARIABLES_GLOBALES_Variable_Ejemplo_VisualBasic_2"
   IOField "Campo ES_5" at 464,170 size 82x32; FormatPattern ????????????????????????????????????????????????????????????????????????????????
      ProcessValue <- "VARIABLES_GLOBALES_variable_string_visual"
   IOField "Campo ES_7" at 334,189 size 107x32; FormatPattern 99999999999999999999
      ProcessValue <- "VARIABLES_GLOBALES_tiempo"

Template "Plantilla_1" 800x420
   Button "Salir" at 720,360 size 78x58; TextOff 'Salir'; PictureOff "ExitRuntime_TP900_Comfort_TR"; PictureOn "ExitRuntime_TP900_Comfort_TR"
      on Release: StopRuntime(0)
   Button "Template_Button" at 640,360 size 78x58; TextOff 'Text'
   Button "Template_Button_1" at 560,360 size 78x58; TextOff 'Text'
   Button "Template_Button_2" at 480,360 size 78x58; TextOff 'Text'
   Button "Template_Button_3" at 400,360 size 78x58; TextOff 'Text'
   Button "Template_Button_4" at 321,360 size 78x58; TextOff 'Text'
   Button "Template_Button_5" at 241,360 size 78x58; TextOff 'Text'
   Button "Template_Button_6" at 161,360 size 78x58; TextOff 'Text'
      on Press: ActivateScreen("Imagen_1", 1)
   Button "Avisos" at 81,360 size 78x58; TextOff 'Avisos'; PictureOff "AlarmDisplay_TP900_Comfort_TR"; PictureOn "AlarmDisplay_TP900_Comfort_TR"
      on Release: function_ef3f5d25("Ventana de avisos_no_acusado", -1)
   Button "Imagen inicial" at 1,360 size 78x58; TextOff 'Imagen inicial'; PictureOff "NavigateHome_TP900_Comfort_TR"; PictureOn "NavigateHome_TP900_Comfort_TR"
      on Release: ActivateScreen("Imagen raíz", 0)

screen "Imagen_1" 800x420, template "Plantilla_1"
   IOField "Plantilla_Campo ES_1" at 178,103 size 73x30; FormatPattern 99999999999999999999
      ProcessValue <- "ALARMAS_DIAS_MOTORES{1}_DIA_HORA_ACTIVACION{1}"
   TextField "Campo de texto_1" at 36,109 size 71x20; Text 'DOMINGO'
   TextField "Campo de texto_2" at 36,142 size 48x20; Text 'LUNES'
   TextField "Campo de texto_3" at 36,176 size 63x20; Text 'MARTES'
   TextField "Campo de texto_4" at 36,210 size 85x20; Text 'MIERCOLES'
   TextField "Campo de texto_5" at 36,243 size 56x20; Text 'JUEVES'
   TextField "Campo de texto_6" at 36,277 size 65x20; Text 'VIERNES'
   TextField "Campo de texto_7" at 36,311 size 65x20; Text 'SABADO'
   TextField "Campo de texto_8" at 140,80 size 140x20; Text 'HORA ACTIVACIÒN'
   TextField "Campo de texto_9" at 270,80 size 167x20; Text 'HORA DESACTIVACION'
   IOField "Plantilla_Campo ES_2" at 307,103 size 73x30; FormatPattern 99999999999999999999
      ProcessValue <- "ALARMAS_DIAS_MOTORES{1}_DIA_HORA_DESACTIVACION{1}"
   IOField "Plantilla_Campo ES_3" at 178,136 size 73x30; FormatPattern 99999999999999999999
      ProcessValue <- "ALARMAS_DIAS_MOTORES{1}_DIA_HORA_ACTIVACION{2}"
   IOField "Plantilla_Campo ES_4" at 307,136 size 73x30; FormatPattern 99999999999999999999
      ProcessValue <- "ALARMAS_DIAS_MOTORES{1}_DIA_HORA_DESACTIVACION{2}"
   IOField "Plantilla_Campo ES_5" at 178,170 size 73x30; FormatPattern 99999999999999999999
      ProcessValue <- "ALARMAS_DIAS_MOTORES{1}_DIA_HORA_ACTIVACION{3}"
   IOField "Plantilla_Campo ES_6" at 307,170 size 73x30; FormatPattern 99999999999999999999
      ProcessValue <- "ALARMAS_DIAS_MOTORES{1}_DIA_HORA_DESACTIVACION{3}"
   IOField "Plantilla_Campo ES_7" at 178,203 size 73x30; FormatPattern 99999999999999999999
      ProcessValue <- "ALARMAS_DIAS_MOTORES{1}_DIA_HORA_ACTIVACION{4}"
   IOField "Plantilla_Campo ES_8" at 307,204 size 73x30; FormatPattern 99999999999999999999
      ProcessValue <- "ALARMAS_DIAS_MOTORES{1}_DIA_HORA_DESACTIVACION{4}"
   IOField "Plantilla_Campo ES_9" at 178,237 size 73x30; FormatPattern 99999999999999999999
      ProcessValue <- "ALARMAS_DIAS_MOTORES{1}_DIA_HORA_ACTIVACION{5}"
   IOField "Plantilla_Campo ES_10" at 307,238 size 73x30; FormatPattern 99999999999999999999
      ProcessValue <- "ALARMAS_DIAS_MOTORES{1}_DIA_HORA_DESACTIVACION{5}"
   IOField "Plantilla_Campo ES_11" at 178,271 size 73x30; FormatPattern 99999999999999999999
      ProcessValue <- "ALARMAS_DIAS_MOTORES{1}_DIA_HORA_ACTIVACION{6}"
   IOField "Plantilla_Campo ES_12" at 307,271 size 73x30; FormatPattern 99999999999999999999
      ProcessValue <- "ALARMAS_DIAS_MOTORES{1}_DIA_HORA_DESACTIVACION{6}"
   IOField "Plantilla_Campo ES_13" at 178,305 size 73x30; FormatPattern 99999999999999999999
      ProcessValue <- "ALARMAS_DIAS_MOTORES{1}_DIA_HORA_ACTIVACION{7}"
   IOField "Plantilla_Campo ES_14" at 307,305 size 73x30; FormatPattern 99999999999999999999
      ProcessValue <- "ALARMAS_DIAS_MOTORES{1}_DIA_HORA_DESACTIVACION{7}"
   GraphicIOField "PlotLight_Round_N_Mono" at 257,55 size 26x26; PictureOn "PilotLight_Round_N_On_mono"; PictureOff "PilotLight_Round_N_Off_mono"
      ProcessValue <- "ALARMAS_DIAS_MOTORES{1}_ESTADO_MOTOR"
   IOField "Plantilla_Campo ES_15" at 468,103 size 73x30; FormatPattern 99999999999999999999
      ProcessValue <- "ALARMAS_DIAS_MOTORES{2}_DIA_HORA_ACTIVACION{1}"
   TextField "Campo de texto_10" at 430,80 size 140x20; Text 'HORA ACTIVACIÒN'
   TextField "Campo de texto_11" at 560,80 size 167x20; Text 'HORA DESACTIVACION'
   IOField "Plantilla_Campo ES_16" at 597,103 size 73x30; FormatPattern 99999999999999999999
      ProcessValue <- "ALARMAS_DIAS_MOTORES{2}_DIA_HORA_DESACTIVACION{1}"
   IOField "Plantilla_Campo ES_17" at 468,136 size 73x30; FormatPattern 99999999999999999999
      ProcessValue <- "ALARMAS_DIAS_MOTORES{2}_DIA_HORA_ACTIVACION{2}"
   IOField "Plantilla_Campo ES_18" at 597,136 size 73x30; FormatPattern 99999999999999999999
      ProcessValue <- "ALARMAS_DIAS_MOTORES{2}_DIA_HORA_DESACTIVACION{2}"
   IOField "Plantilla_Campo ES_19" at 468,170 size 73x30; FormatPattern 99999999999999999999
      ProcessValue <- "ALARMAS_DIAS_MOTORES{2}_DIA_HORA_ACTIVACION{3}"
   IOField "Plantilla_Campo ES_20" at 597,170 size 73x30; FormatPattern 99999999999999999999
      ProcessValue <- "ALARMAS_DIAS_MOTORES{2}_DIA_HORA_DESACTIVACION{3}"
   IOField "Plantilla_Campo ES_21" at 468,203 size 73x30; FormatPattern 99999999999999999999
      ProcessValue <- "ALARMAS_DIAS_MOTORES{2}_DIA_HORA_ACTIVACION{4}"
   IOField "Plantilla_Campo ES_22" at 597,204 size 73x30; FormatPattern 99999999999999999999
      ProcessValue <- "ALARMAS_DIAS_MOTORES{2}_DIA_HORA_DESACTIVACION{4}"
   IOField "Plantilla_Campo ES_23" at 468,237 size 73x30; FormatPattern 99999999999999999999
      ProcessValue <- "ALARMAS_DIAS_MOTORES{2}_DIA_HORA_ACTIVACION{5}"
   IOField "Plantilla_Campo ES_24" at 597,238 size 73x30; FormatPattern 99999999999999999999
      ProcessValue <- "ALARMAS_DIAS_MOTORES{2}_DIA_HORA_DESACTIVACION{5}"
   IOField "Plantilla_Campo ES_25" at 468,271 size 73x30; FormatPattern 99999999999999999999
      ProcessValue <- "ALARMAS_DIAS_MOTORES{2}_DIA_HORA_ACTIVACION{6}"
   IOField "Plantilla_Campo ES_26" at 597,271 size 73x30; FormatPattern 99999999999999999999
      ProcessValue <- "ALARMAS_DIAS_MOTORES{2}_DIA_HORA_DESACTIVACION{6}"
   IOField "Plantilla_Campo ES_27" at 468,305 size 73x30; FormatPattern 99999999999999999999
      ProcessValue <- "ALARMAS_DIAS_MOTORES{2}_DIA_HORA_ACTIVACION{7}"
   IOField "Plantilla_Campo ES_28" at 597,305 size 73x30; FormatPattern 99999999999999999999
      ProcessValue <- "ALARMAS_DIAS_MOTORES{2}_DIA_HORA_DESACTIVACION{7}"
   GraphicIOField "PlotLight_Round_N_Mono_1" at 547,55 size 26x26; PictureOff "PilotLight_Round_N_Off_mono"; PictureOn "PilotLight_Round_N_On_mono"
      ProcessValue <- "ALARMAS_DIAS_MOTORES{2}_ESTADO_MOTOR"

VB script "FuncionVB_1"
   'Sugerencia:
   ' 1. Utilice la combinación de teclas <CTRL+ESPACIO> o <CTRL+I> para abrir una lista de todos los objetos y funciones
   ' 2. Escriba el código utilizando el objeto HMI Runtime.
   '  Ejemplo: HmiRuntime.Screens("Screen_1").
   ' 3. Utilice la combinación de teclas <CTRL+J> para crear una referencia de objeto..
   'Escriba el código a partir de esta posición:
   'VARIABLES_GLOBALES_Variable_Ejemplo_VisualBasic_2=23
   SmartTags("VARIABLES_GLOBALES_Variable_Ejemplo_VisualBasic_2")=13
   SmartTags("VARIABLES_GLOBALES_variable_string_visual")="ALFREDO"
   SmartTags("VARIABLES_GLOBALES_variable_string_visual2{0}")="PUTA LETY"

VB script "FuncionVB_2"
   'Sugerencia:
   ' 1. Utilice la combinación de teclas <CTRL+ESPACIO> o <CTRL+I> para abrir una lista de todos los objetos y funciones
   ' 2. Escriba el código utilizando el objeto HMI Runtime.
   '  Ejemplo: HmiRuntime.Screens("Screen_1").
   ' 3. Utilice la combinación de teclas <CTRL+J> para crear una referencia de objeto..
   'Escriba el código a partir de esta posición:
   
   FuncionVB_2=Parametro_1+Parametro_2
*)